KUKA KRL data list: braketestreq.dat

&ACCESS RV
&REL 1
&COMMENT BrkTst-main task
&PARAM EDITMASK = *
DEFDAT  BRAKETESTREQ
;FOLD EXTERNAL DECLARATIONS;%{PE}%MKUKATPBASIS,%CEXT,%VCOMMON,%P
;FOLD BASISTECH EXT;%{PE}%MKUKATPBASIS,%CEXT,%VEXT,%P
EXT  BAS (BAS_COMMAND  :IN,REAL  :IN )
DECL INT SUCCESS
;ENDFOLD (BASISTECH EXT)
;FOLD USER EXT;%{E}%MKUKATPUSER,%CEXT,%VEXT,%P
;ENDFOLD (USER EXT)
;ENDFOLD (EXTERNAL DECLERATIONS)
INT AxNr, BtIrNr
INT PerformBrakeTest=0; index for $flag to trigger brake test
ENDDAT
